(* LS Electric XG5000 project: XEM_L7P_ModRTU_Example *)
(* PLC LSPLC *)
(* module base 0 slot 0: Input/Output Module:XEM-DN/DP32HP (DC 24V Input, Transistor Output, 32 Contacts) *)
(* module base 0 slot 1: Internal Positioning:XBF-PO06E (Open Collector Type, 6 Axis) *)
VAR_GLOBAL
    gIndex01_Distance AT %MW10 : ARRAY[0..1] OF WORD; (* global word data to change Index01 distance value. *)
    gIndex01_IndexType AT %MW12 : WORD; (* global word data to change Index01 index type *)
    gMotion_Start AT %MX1 : BOOL; (* global command to start index movement sent over Modbus RTU *)
    gSV_ON AT %MX0 : BOOL; (* global Command to turn servo on/off sent over Modbus RTU *)
    ISEL0 AT %MX2 : BOOL; (* ISEL0 of L7P *)
    ISEL1 AT %MX3 : BOOL; (* ISEL1 of L7P *)
    ISEL2 AT %MX4 : BOOL; (* ISEL2 of L7P *)
    ISEL3 AT %MX5 : BOOL; (* ISEL3 of L7P *)
    ISEL4 AT %MX6 : BOOL; (* ISEL4 of L7P *)
    ISEL5 AT %MX7 : BOOL; (* ISEL5 of L7P *)
END_VAR

PROGRAM NewProgram (* task: Scan Program *)
VAR_EXTERNAL
    gIndex01_Distance : ARRAY[0..1] OF WORD; (* AT %MW10 *) (* global word data to change Index01 distance value. *)
    gIndex01_IndexType : WORD; (* AT %MW12 *) (* global word data to change Index01 index type *)
    gMotion_Start : BOOL; (* AT %MX1 *) (* global command to start index movement sent over Modbus RTU *)
    gSV_ON : BOOL; (* AT %MX0 *) (* global Command to turn servo on/off sent over Modbus RTU *)
    ISEL0 : BOOL; (* AT %MX2 *) (* ISEL0 of L7P *)
    ISEL1 : BOOL; (* AT %MX3 *) (* ISEL1 of L7P *)
    ISEL2 : BOOL; (* AT %MX4 *) (* ISEL2 of L7P *)
    ISEL3 : BOOL; (* AT %MX5 *) (* ISEL3 of L7P *)
    ISEL4 : BOOL; (* AT %MX6 *) (* ISEL4 of L7P *)
    ISEL5 : BOOL; (* AT %MX7 *) (* ISEL5 of L7P *)
END_VAR
VAR
    Index : USINT; (* Index in decimal form.  will be converted to bit form *)
    Index01_Distance : DINT; (* local index01 distance value *)
    Index01_Index_Type : WORD; (* local index01 type *)
    Servo_Enable : BOOL; (* Enable servo - local command to enable servos *)
    Start_Motion : BOOL; (* local command to start motion *)
    tempDword : DWORD; (* temporary dword storage *)
END_VAR

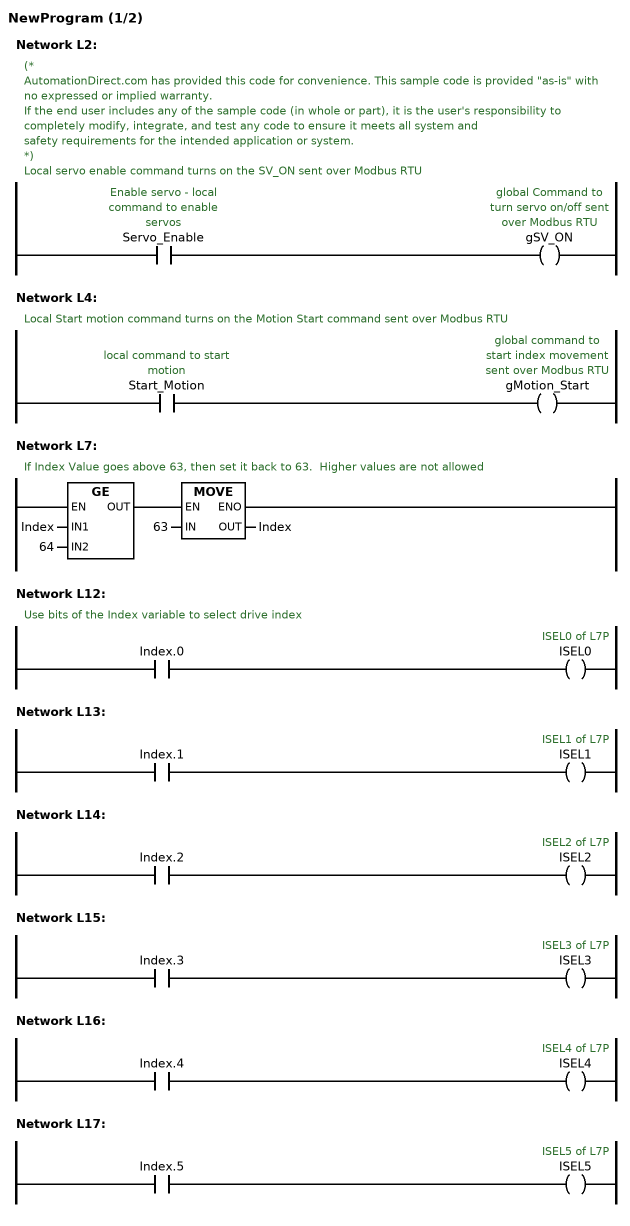
(* ( * / AutomationDirect.com has provided this code for convenience. This sample code is provided "as-is" with no expressed or implied warranty. / If the end user includes any of the sample code (in whole or part), it is the user's responsibility to completely modify, integrate, and test any code to ensure it meets all system and / safety requirements for the intended application or system. / * ) *)
(* Local servo enable command turns on the SV_ON sent over Modbus RTU *)
(* Rung L2 *)
gSV_ON := Servo_Enable;
(* Local Start motion command turns on the Motion Start command sent over Modbus RTU *)
(* Rung L4 *)
gMotion_Start := Start_Motion;
(* If Index Value goes above 63, then set it back to 63.  Higher values are not allowed *)
(* Rung L7 *)
IF Index >= 64 THEN Index := 63; END_IF;
(* Use bits of the Index variable to select drive index *)
(* Rung L12 *)
ISEL0 := Index.0;
(* Rung L13 *)
ISEL1 := Index.1;
(* Rung L14 *)
ISEL2 := Index.2;
(* Rung L15 *)
ISEL3 := Index.3;
(* Rung L16 *)
ISEL4 := Index.4;
(* Rung L17 *)
ISEL5 := Index.5;

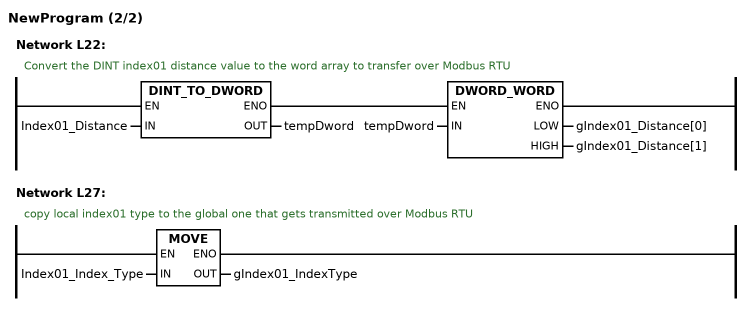
(* Convert the DINT index01 distance value to the word array to transfer over Modbus RTU *)
(* Rung L22 *)
tempDword := DINT_TO_DWORD(Index01_Distance);
gIndex01_Distance[0] := DWORD_WORD(IN := tempDword, HIGH => gIndex01_Distance[1]);
(* copy local index01 type to the global one that gets transmitted over Modbus RTU *)
(* Rung L27 *)
gIndex01_IndexType := Index01_Index_Type;
END_PROGRAM